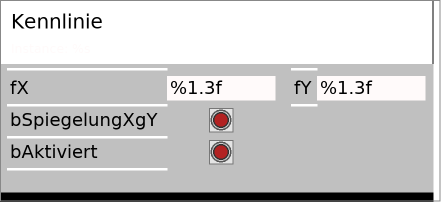
VISUALIZATION RET_VISU_Kennlinie  // 441x202
VAR_INPUT
   {attribute 'parameterstringof' := 'm_Input_FB'}
   m_Input_INST_Str : STRING;
END_VAR
VAR_IN_OUT
   m_Input_FB : Kennlinie;
END_VAR
    RoundedRectangle (0,0 433x81)
    RoundedRectangle (0,162 433x40)
    Rectangle (0,64 433x128)
    PushSwitch (209,108 24x24), variable: m_Input_FB.bSpiegelungXgY, behaviour: TOGGLE, style: Switch-PushSwitch-Red
    PushSwitch (209,140 24x24), variable: m_Input_FB.bAktiviert, behaviour: TOGGLE, style: Switch-PushSwitch-Red
    Rectangle (8,8 433x27), "Kennlinie"
    Rectangle (8,35 433x27), "Instance: %s", text variable: m_Input_INST_Str
    Rectangle (7,68 160x2)
    Rectangle (167,76 108x24), "%1.3f", text variable: m_Input_FB.fX
        OnMouseClick: write the text variable via Default
    Rectangle (7,76 160x24), "fX"
    Rectangle (7,104 160x2)
    Rectangle (7,108 160x24), "bSpiegelungXgY"
    Rectangle (7,136 160x2)
    Rectangle (7,140 160x24), "bAktiviert"
    Rectangle (7,168 160x2)
    Rectangle (291,68 26x2)
    Rectangle (317,76 108x24), "%1.3f", text variable: m_Input_FB.fY
    Rectangle (291,76 26x24), "fY"
    Rectangle (291,104 26x2)
END_VISUALIZATION

(* stored: Version 1.1.0.1, ProductVersion 3.1.4024.12
   Visu RET_VISU_Kennlinie: Id {f5a03ef4-98e6-4fcc-8285-374d9dae0e03} *)
